FUNCTION_BLOCK SET_LINE_DATA (* Sets line data to the proper format before sending to machine *)
  (* Standard: 61499-2 *)
  (* Version 1.0, 17-04-2012, GASR, Universidade do Estado de Santa Catarina *)
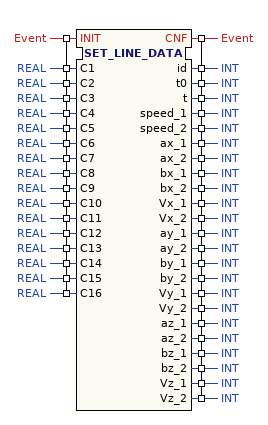
  EVENT_INPUT
    INIT WITH C1, C2, C3, C4, C5, C6, C7, C8, C9, C10, C11, C12, C13, C14, C15, C16;
  END_EVENT
  EVENT_OUTPUT
    CNF WITH id, t0, t, speed_1, speed_2, ax_1, ax_2, bx_1, bx_2, Vx_1, Vx_2, ay_1, ay_2, by_1, by_2, Vy_1, Vy_2, az_1, az_2, bz_1, bz_2, Vz_1, Vz_2;
  END_EVENT
  VAR_INPUT
    C1 : REAL; (* Coeficient 1 *)
    C2 : REAL; (* Coeficient 2 *)
    C3 : REAL; (* Coeficient 3 *)
    C4 : REAL; (* Coeficient 4 *)
    C5 : REAL; (* Coeficient 5 *)
    C6 : REAL; (* Coeficient 6 *)
    C7 : REAL; (* Coeficient 7 *)
    C8 : REAL; (* Coeficient 8 *)
    C9 : REAL; (* Coeficient 9 *)
    C10 : REAL; (* Coeficient 10 *)
    C11 : REAL; (* Coeficient 11 *)
    C12 : REAL; (* Coeficient 12 *)
    C13 : REAL; (* Coeficient 13 *)
    C14 : REAL; (* Coeficient 14 *)
    C15 : REAL; (* Coeficient 15 *)
    C16 : REAL; (* Coeficient 16 *)
  END_VAR
  VAR_OUTPUT
    id : INT;
    t0 : INT;
    t : INT;
    speed_1 : INT;
    speed_2 : INT;
    ax_1 : INT;
    ax_2 : INT;
    bx_1 : INT;
    bx_2 : INT;
    Vx_1 : INT;
    Vx_2 : INT;
    ay_1 : INT;
    ay_2 : INT;
    by_1 : INT;
    by_2 : INT;
    Vy_1 : INT;
    Vy_2 : INT;
    az_1 : INT;
    az_2 : INT;
    bz_1 : INT;
    bz_2 : INT;
    Vz_1 : INT;
    Vz_2 : INT;
  END_VAR
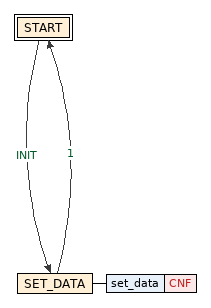
  EC_STATES
    START;
    SET_DATA : set_data -> CNF;
  END_STATES
  EC_TRANSITIONS
    START TO SET_DATA := INIT;
    SET_DATA TO START := 1;
  END_TRANSITIONS
  ALGORITHM set_data IN Lua:
function float_to_ints( n, precision )
	local n_1, n_2
	if( tonumber(n) >= 0 ) then
		n_1 = math.floor( n )
		n_2 = (n - n_1)*(10^precision)
		n_2 = math.floor( n_2 )
	else
		n_1 = math.ceil( n )
		n_2 = (n - n_1)*(10^precision)
		n_2 = math.ceil( n_2 )
	end
	return n_1, n_2
end

id = C1
t0 = C8
t = C9
print( 'Feed = ', C13 )
C13 = (C13/0.005)*60
print( 'Feed = ', C13 )
C14 = math.abs( C14 )
C15 = math.abs( C15 )
C16 = math.abs( C16 )
speed_1, speed_2 = float_to_ints( C13, 3 )
ax_1, ax_2 = float_to_ints( C2, 3 )
bx_1, bx_2 = float_to_ints( C5, 3 )
Vx_1, Vx_2 = float_to_ints( C14, 3 )
ay_1, ay_2 = float_to_ints( C3, 3 )
by_1, by_2 = float_to_ints( C6, 3 )
Vy_1, Vy_2 = float_to_ints( C15, 3 )
az_1, az_2 = float_to_ints( C4, 3 )
bz_1, bz_2 = float_to_ints( C7, 3 )
Vz_1, Vz_2 = float_to_ints( C16, 3 )
  END_ALGORITHM
END_FUNCTION_BLOCK
